// TIA Portal V20 export
ORGANIZATION_BLOCK "HardwareInterrupt"   // OB40, LAD, HardwareInterrupt
// stored: SetENOAutomatically false
   VAR_INPUT
      LADDR : HW_IO;   // Hardware identifier
      USI : Word;   // User structure identifier
      IChannel : USInt;   // Interrupt channel number
      EventType : Byte;   // EventType
      PointAddr : DWord;
   END_VAR
BEGIN
END_ORGANIZATION_BLOCK
